FUNCTION_BLOCK SS3_ifb_Vaccume_Gripper (* Basic FB with empty ECC *)
  (* Standard: 61499-2 *)
  (* Version 1.0, 2021-08-23, AK121668 *)
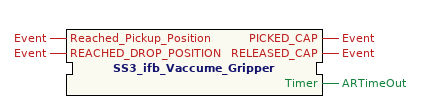
  EVENT_INPUT
    Reached_Pickup_Position;
    REACHED_DROP_POSITION;
  END_EVENT
  EVENT_OUTPUT
    PICKED_CAP;
    RELEASED_CAP;
  END_EVENT
  PLUGS
    Timer : ARTimeOut;
  END_PLUGS
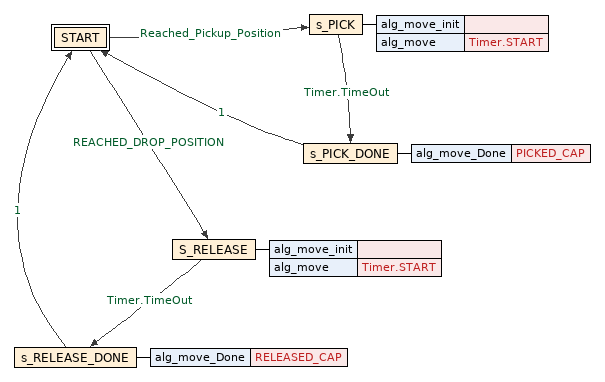
  EC_STATES
    START; (* Initial State *)
    s_PICK : alg_move_init, alg_move -> Timer.START;
    s_PICK_DONE : alg_move_Done -> PICKED_CAP;
    S_RELEASE : alg_move_init, alg_move -> Timer.START;
    s_RELEASE_DONE : alg_move_Done -> RELEASED_CAP;
  END_STATES
  EC_TRANSITIONS
    s_PICK_DONE TO START := 1;
    START TO s_PICK := Reached_Pickup_Position;
    s_PICK TO s_PICK_DONE := Timer.TimeOut;
    s_RELEASE_DONE TO START := 1;
    START TO S_RELEASE := REACHED_DROP_POSITION;
    S_RELEASE TO s_RELEASE_DONE := Timer.TimeOut;
  END_TRANSITIONS
  ALGORITHM alg_move_init IN ST:
Timer.DT := T#3s;
  END_ALGORITHM
  ALGORITHM alg_move IN ST:

  END_ALGORITHM
  ALGORITHM alg_move_Done IN ST:

  END_ALGORITHM
END_FUNCTION_BLOCK
